// TwinCAT 3 PLC project PlcProjekt
// ProgramVersion: 3.1.4023.0
// libraries:
//   Tc2_Standard, * (Beckhoff Automation GmbH)
//   Tc2_System, * (Beckhoff Automation GmbH)
//   Tc3_Module, * (Beckhoff Automation GmbH)
// project tree:
//   GVLs/ DaDi.TcGVL
//   / PlcTask.TcTTO
//   POUs/ EinProgramm.TcPOU, MAIN.TcPOU
// real-time tasks:
//   TASK PlcTask: cycle T#10ms, priority 20, ADS port 350
// motion (NC):
//   TASK NC-Task 1 SAF: cycle T#2ms, priority 4, ADS port 501
//   TASK NC-Task 1 SVB: cycle T#10ms, priority 8, ADS port 511
//   AXIS Achse 1: X-Achse (id 1)
//     OtherSettings: AllowMotionCmdToSlave=true
//     encoder EncType=19
//       EncPara: MaxCount=#xffffffff
//     drive DrvType=16
//       DrvPara: MaxCount=#xffffffff, DriveControlDWord=#x00020000
//         Analog: TorqueSetpointScale=10, ScaleFactorActTorque=0.1
//         TimeComp: TaskDelayCycles=1
//     controller CtrType=1
//       CtrPara: PriorControlFactor=1
//         Observer: BandWidth=20
//   AXIS Achse 2: Y-Achse (id 2)
//     OtherSettings: AllowMotionCmdToSlave=true
//     encoder EncType=19
//       EncPara: MaxCount=#xffffffff
//     drive DrvType=16
//       DrvPara: MaxCount=#xffffffff, DriveControlDWord=#x00020000
//         Analog: TorqueSetpointScale=10, ScaleFactorActTorque=0.1
//         TimeComp: TaskDelayCycles=1
//     controller CtrType=1
//       CtrPara: PriorControlFactor=1
//         Observer: BandWidth=20
//   AXIS Achse 3: Z-Achse (id 3)
//     OtherSettings: AllowMotionCmdToSlave=true
//     encoder EncType=4
//       EncPara: MaxCount=#x0000ffff
//         Inc: RefSoftSyncMask=#x0000ffff
//     drive DrvType=24
//       Analog: TorqueSetpointScale=10, ScaleFactorActTorque=0.1
//       TimeComp: TaskDelayCycles=1
//     controller CtrType=1
//       CtrPara: PriorControlFactor=1
//         Observer: BandWidth=20
//   AXIS Achse 4 (id 4)
//     OtherSettings: AllowMotionCmdToSlave=true
//     encoder EncType=4
//       EncPara: MaxCount=#x0000ffff
//     drive DrvType=23
//       Analog: TorqueSetpointScale=10, ScaleFactorActTorque=0.1
//       TimeComp: TaskDelayCycles=1
//     controller CtrType=1
//       CtrPara: PriorControlFactor=1
//         Observer: BandWidth=20
//   AXIS Achse 5 (id 5)
//     OtherSettings: AllowMotionCmdToSlave=true
//     encoder EncType=4
//       EncPara: MaxCount=#x0000ffff
//     drive DrvType=23
//       Analog: TorqueSetpointScale=10, ScaleFactorActTorque=0.1
//       TimeComp: TaskDelayCycles=1
//     controller CtrType=1
//       CtrPara: PriorControlFactor=1
//         Observer: BandWidth=20
// I/O:
//   DEVICE Gerät 1 (EtherCAT), AmsNetId 5.99.63.148.2.1
//     Klemme 1 (EK1200) [EK1200-5000 EtherCAT Netzteil (2A E-Bus)]
//       Klemme 2 (EL1859) [EL1859 8K. Dig. Eingang 24V, 3ms, 8K. Dig. Ausgang 24V, 0.5A]
//       Klemme 3 (EL7201-0010): X-Achse [EL7201-0010 1K. MDP742 Servo-Motor-Endstufe mit OCT (50V, 2,8A RMS)]
//       Klemme 4 (EL7201-0010): Y-Achse [EL7201-0010 1K. MDP742 Servo-Motor-Endstufe mit OCT (50V, 2,8A RMS)]
//       Klemme 5 (EL7037): Z-Achse [EL7037 1K. Schrittmotor-Endstufe (24V, 1.5A)]
//       Klemme 6 (EL7332): DC-Motor [EL7332 2K. DC-Motor-Endstufe (24V, 1.5A)]
//       Klemme 7 (EL9011) [EL9011 Endklemme]
// variable links:
//   NC-Task 1 SAF/Axes/Achse 1: X-Achse <-> Device 1 (EtherCAT)/Term 1 (EK1200)/Klemme 3 (EL7201-0010): X-Achse
//     Drive/Inputs/In/nDcOutputTime <-> InfoData/DcOutputShift
//     Drive/Inputs/In/nState1 <-> DRV Statusword/Statusword
//     Drive/Inputs/In/nState2 <-> DRV Statusword/Statusword @bit 8
//     Drive/Inputs/In/nState4 @bit 1 <-> WcState/InputToggle
//     Drive/Inputs/In/nState4 <-> WcState/WcState
//     Drive/Outputs/Out/nCtrl1 <-> DRV Controlword/Controlword
//     Drive/Outputs/Out/nCtrl2 <-> DRV Controlword/Controlword @bit 8
//     Drive/Outputs/Out/nDataOut2 <-> DRV Target velocity/Target velocity
//     Enc/Inputs/In/nDataIn1 <-> FB Position/Position
//     Enc/Inputs/In/nDcInputTime <-> InfoData/DcInputShift
//     Enc/Inputs/In/nState4 @bit 1 <-> WcState/InputToggle
//     Enc/Inputs/In/nState4 <-> WcState/WcState
//   NC-Task 1 SAF/Axes/Achse 2: Y-Achse <-> Device 1 (EtherCAT)/Term 1 (EK1200)/Klemme 4 (EL7201-0010): Y-Achse
//     Drive/Inputs/In/nDcOutputTime <-> InfoData/DcOutputShift
//     Drive/Inputs/In/nState1 <-> DRV Statusword/Statusword
//     Drive/Inputs/In/nState2 <-> DRV Statusword/Statusword @bit 8
//     Drive/Inputs/In/nState4 @bit 1 <-> WcState/InputToggle
//     Drive/Inputs/In/nState4 <-> WcState/WcState
//     Drive/Outputs/Out/nCtrl1 <-> DRV Controlword/Controlword
//     Drive/Outputs/Out/nCtrl2 <-> DRV Controlword/Controlword @bit 8
//     Drive/Outputs/Out/nDataOut2 <-> DRV Target velocity/Target velocity
//     Enc/Inputs/In/nDataIn1 <-> FB Position/Position
//     Enc/Inputs/In/nDcInputTime <-> InfoData/DcInputShift
//     Enc/Inputs/In/nState4 @bit 1 <-> WcState/InputToggle
//     Enc/Inputs/In/nState4 <-> WcState/WcState
//   NC-Task 1 SAF/Axes/Achse 3: Z-Achse <-> Device 1 (EtherCAT)/Term 1 (EK1200)/Klemme 5 (EL7037): Z-Achse
//     Drive/Inputs/In/nState1 @bit 3 <-> STM Status/Status/Error
//     Drive/Inputs/In/nState1 @bit 7 <-> STM Status/Status/Motor stall
//     Drive/Inputs/In/nState1 @bit 5 <-> STM Status/Status/Moving negative
//     Drive/Inputs/In/nState1 @bit 4 <-> STM Status/Status/Moving positive
//     Drive/Inputs/In/nState1 @bit 1 <-> STM Status/Status/Ready
//     Drive/Inputs/In/nState1 <-> STM Status/Status/Ready to enable
//     Drive/Inputs/In/nState1 @bit 6 <-> STM Status/Status/Torque reduced
//     Drive/Inputs/In/nState1 @bit 2 <-> STM Status/Status/Warning
//     Drive/Inputs/In/nState2 @bit 3 <-> STM Status/Status/Digital input 1
//     Drive/Inputs/In/nState2 @bit 4 <-> STM Status/Status/Digital input 2
//     Drive/Inputs/In/nState2 @bit 5 <-> STM Status/Status/Sync error
//     Drive/Inputs/In/nState2 @bit 7 <-> STM Status/Status/TxPDO Toggle
//     Drive/Inputs/In/nState4 @bit 1 <-> WcState/InputToggle
//     Drive/Inputs/In/nState4 <-> WcState/WcState
//     Drive/Outputs/Out/nCtrl1 <-> STM Control/Control/Enable
//     Drive/Outputs/Out/nCtrl1 @bit 2 <-> STM Control/Control/Reduce torque
//     Drive/Outputs/Out/nCtrl1 @bit 1 <-> STM Control/Control/Reset
//     Drive/Outputs/Out/nCtrl2 @bit 3 <-> STM Control/Control/Digital output 1
//     Drive/Outputs/Out/nDataOut2[0] <-> STM Velocity/Velocity
//     Enc/Inputs/In/nDataIn1[0] <-> ENC Status compact/Counter value
//     Enc/Inputs/In/nDataIn2[0] <-> ENC Status compact/Latch value
//     Enc/Inputs/In/nState1 @bit 4 <-> ENC Status compact/Status/Counter overflow
//     Enc/Inputs/In/nState1 @bit 3 <-> ENC Status compact/Status/Counter underflow
//     Enc/Inputs/In/nState1 @bit 7 <-> ENC Status compact/Status/Extrapolation stall
//     Enc/Inputs/In/nState1 <-> ENC Status compact/Status/Latch C valid
//     Enc/Inputs/In/nState1 @bit 1 <-> ENC Status compact/Status/Latch extern valid
//     Enc/Inputs/In/nState1 @bit 2 <-> ENC Status compact/Status/Set counter done
//     Enc/Inputs/In/nState2 @bit 4 <-> ENC Status compact/Status/Status of extern latch
//     Enc/Inputs/In/nState2 <-> ENC Status compact/Status/Status of input A
//     Enc/Inputs/In/nState2 @bit 1 <-> ENC Status compact/Status/Status of input B
//     Enc/Inputs/In/nState2 @bit 2 <-> ENC Status compact/Status/Status of input C
//     Enc/Inputs/In/nState2 @bit 5 <-> ENC Status compact/Status/Sync error
//     Enc/Inputs/In/nState2 @bit 7 <-> ENC Status compact/Status/TxPDO Toggle
//     Enc/Inputs/In/nState4 @bit 1 <-> WcState/InputToggle
//     Enc/Inputs/In/nState4 <-> WcState/WcState
//     Enc/Outputs/Out/nCtrl1 <-> ENC Control compact/Control/Enable latch C
//     Enc/Outputs/Out/nCtrl1 @bit 3 <-> ENC Control compact/Control/Enable latch extern on negative edge
//     Enc/Outputs/Out/nCtrl1 @bit 1 <-> ENC Control compact/Control/Enable latch extern on positive edge
//     Enc/Outputs/Out/nCtrl1 @bit 2 <-> ENC Control compact/Control/Set counter
//     Enc/Outputs/Out/nDataOut1[0] <-> ENC Control compact/Set counter value
//   NC-Task 1 SAF/Axes/Achse 4 <-> Device 1 (EtherCAT)/Term 1 (EK1200)/Klemme 6 (EL7332): DC-Motor
//     Drive/Inputs/In/nState1 @bit 3 <-> DCM Status Channel 1/Status/Error
//     Drive/Inputs/In/nState1 @bit 5 <-> DCM Status Channel 1/Status/Moving negative
//     Drive/Inputs/In/nState1 @bit 4 <-> DCM Status Channel 1/Status/Moving positive
//     Drive/Inputs/In/nState1 @bit 1 <-> DCM Status Channel 1/Status/Ready
//     Drive/Inputs/In/nState1 <-> DCM Status Channel 1/Status/Ready to enable
//     Drive/Inputs/In/nState1 @bit 6 <-> DCM Status Channel 1/Status/Torque reduced
//     Drive/Inputs/In/nState1 @bit 2 <-> DCM Status Channel 1/Status/Warning
//     Drive/Inputs/In/nState2 @bit 3 <-> DCM Status Channel 1/Status/Digital input 1
//     Drive/Inputs/In/nState2 @bit 4 <-> DCM Status Channel 1/Status/Digital input 2
//     Drive/Inputs/In/nState2 @bit 5 <-> DCM Status Channel 1/Status/Sync error
//     Drive/Inputs/In/nState2 @bit 7 <-> DCM Status Channel 1/Status/TxPDO Toggle
//     Drive/Inputs/In/nState4 @bit 1 <-> WcState/InputToggle
//     Drive/Inputs/In/nState4 <-> WcState/WcState
//     Drive/Outputs/Out/nCtrl1 <-> DCM Control Channel 1/Control/Enable
//     Drive/Outputs/Out/nCtrl1 @bit 2 <-> DCM Control Channel 1/Control/Reduce torque
//     Drive/Outputs/Out/nCtrl1 @bit 1 <-> DCM Control Channel 1/Control/Reset
//     Drive/Outputs/Out/nDataOut2[0] <-> DCM Velocity Channel 1/Velocity
//   NC-Task 1 SAF/Axes/Achse 5 <-> Device 1 (EtherCAT)/Term 1 (EK1200)/Klemme 6 (EL7332): DC-Motor
//     Drive/Inputs/In/nState1 @bit 3 <-> DCM Status Channel 2/Status/Error
//     Drive/Inputs/In/nState1 @bit 5 <-> DCM Status Channel 2/Status/Moving negative
//     Drive/Inputs/In/nState1 @bit 4 <-> DCM Status Channel 2/Status/Moving positive
//     Drive/Inputs/In/nState1 @bit 1 <-> DCM Status Channel 2/Status/Ready
//     Drive/Inputs/In/nState1 <-> DCM Status Channel 2/Status/Ready to enable
//     Drive/Inputs/In/nState1 @bit 6 <-> DCM Status Channel 2/Status/Torque reduced
//     Drive/Inputs/In/nState1 @bit 2 <-> DCM Status Channel 2/Status/Warning
//     Drive/Inputs/In/nState2 @bit 3 <-> DCM Status Channel 2/Status/Digital input 1
//     Drive/Inputs/In/nState2 @bit 4 <-> DCM Status Channel 2/Status/Digital input 2
//     Drive/Inputs/In/nState2 @bit 5 <-> DCM Status Channel 2/Status/Sync error
//     Drive/Inputs/In/nState2 @bit 7 <-> DCM Status Channel 2/Status/TxPDO Toggle
//     Drive/Inputs/In/nState4 @bit 1 <-> WcState/InputToggle
//     Drive/Inputs/In/nState4 <-> WcState/WcState
//     Drive/Outputs/Out/nCtrl1 <-> DCM Control Channel 2/Control/Enable
//     Drive/Outputs/Out/nCtrl1 @bit 2 <-> DCM Control Channel 2/Control/Reduce torque
//     Drive/Outputs/Out/nCtrl1 @bit 1 <-> DCM Control Channel 2/Control/Reset
//     Drive/Outputs/Out/nDataOut2[0] <-> DCM Velocity Channel 2/Velocity
//   PlcProjekt/PlcProjekt Instance <-> Device 1 (EtherCAT)/Term 1 (EK1200)/Term 2 (EL1859)
//     PlcTask Inputs/DaDi.B{1..8} <-> Channel {1..8}/Input  (8 links)
//     PlcTask Outputs/DaDi.P{1..8} <-> Channel {9..16}/Output  (8 links)

CONFIGURATION PlcProjekt
    RESOURCE PLC ON TwinCAT3
        TASK PlcTask(INTERVAL := T#10ms, PRIORITY := 20);
        PROGRAM MAIN WITH PlcTask : MAIN;
    END_RESOURCE
END_CONFIGURATION

// ---- GVLs/DaDi.TcGVL
{attribute 'qualified_only'}
VAR_GLOBAL
	B1 AT %I*: BOOL;
	B2 AT %I*: BOOL;
	B3 AT %I*: BOOL;
	B4 AT %I*: BOOL;
	B5 AT %I*: BOOL;
	B6 AT %I*: BOOL;
	B7 AT %I*: BOOL;
	B8 AT %I*: BOOL;

	P1 AT %Q*: BOOL;
	P2 AT %Q*: BOOL;
	P3 AT %Q*: BOOL;
	P4 AT %Q*: BOOL;
	P5 AT %Q*: BOOL;
	P6 AT %Q*: BOOL;
	P7 AT %Q*: BOOL;
	P8 AT %Q*: BOOL;	
END_VAR

// ---- POUs/MAIN.TcPOU
PROGRAM MAIN
VAR	
END_VAR

EinProgramm();

END_PROGRAM

// ---- POUs/EinProgramm.TcPOU
PROGRAM EinProgramm
VAR
	Timer1: TON;
	Timer2: TON;
END_VAR

DaDi.P1:=DaDi.B1;
DaDi.P2:=DaDi.B2;
DaDi.P3:=DaDi.B3;
DaDi.P4:=DaDi.B4;
(*
DaDi.P5:=DaDi.B5;
DaDi.P6:=DaDi.B6;
DaDi.P7:=DaDi.B7;
DaDi.P8:=DaDi.B8;
*)
Timer1(IN:=NOT Timer2.Q, Pt:=T#200MS);
Timer2(IN:= Timer1.Q, PT:= T#200MS);

DaDi.P7:= NOT Timer1.Q;
DaDi.P8:= Timer1.Q;

END_PROGRAM
